// This function has been automatically generated from the project information.
{attribute 'signature_flag' := '1073741824'}
{attribute 'TcGenerated'}
{attribute 'no-analysis'}
FUNCTION F_GetTitle : WSTRING
VAR_INPUT
	
END_VAR

F_GetTitle := "FsError";

END_FUNCTION

(* stored: Version 1.1.0.1
   POU F_GetTitle: Id {7315f40d-68bf-022f-1431-1cc6aa71c035}, SpecialFunc None *)
